FUNCTION_BLOCK FB_MotionAxisMoveAbsoluteSmaract IMPLEMENTS I_MotionAxisMoveAbsolute
VAR
END_VAR

END_FUNCTION_BLOCK

(* stored: Version 1.1.0.1
   POU FB_MotionAxisMoveAbsoluteSmaract: Id {ec5c3586-237a-4aa3-9c3f-c43958cba9ce}, SpecialFunc None *)
